// TIA Portal V17 export
// export: Created 2026-04-13T11:12:53.8543226Z, ExportSetting WithDefaults, DisplayName Totally Integrated Automation Portal, DisplayVersion V17 Update 4, DisplayName TIA Portal Openness, DisplayVersion V17 Update 4, DisplayName TIA Portal Version Control Interface, DisplayVersion V17, DisplayName SINAMICS Startdrive Advanced, DisplayVersion V17, DisplayName SINAMICS Startdrive G130, G150, S120, S150, SINAMICS MV, S210, DisplayVersion V17, DisplayName SINAMICS Startdrive G110M, G120, G120C, G120D, G120P, G115D, DisplayVersion V17, DisplayName STEP 7 Professional, DisplayVersion V17 Update 4, DisplayName STEP 7 Safety, DisplayVersion V17, DisplayName WinCC Professional, DisplayVersion V17 Update 4
TagTable "PW"
  PW_PH批号输入 : Int  (PLC tag PW.PH批号输入, HMI_连接_1, 1 s)
  PW_MS模式设定 : Real  (PLC tag PW.MS模式设定, HMI_连接_1, 1 s)
  PW_AQ安全停机 : Bool  (PLC tag PW.AQ安全停机, HMI_连接_1, 1 s)
  PW_自动运行报警 : Bool  (PLC tag PW.自动运行报警, HMI_连接_1, 1 s)
  PW_自动停止 : Bool  (PLC tag PW.自动停止, HMI_连接_1, 1 s)
  PW_MS模式状态 : Int  (PLC tag PW.MS模式状态, HMI_连接_1, 1 s)
  PW_ZT总通路 : Int  (PLC tag PW.ZT总通路, HMI_连接_1, 1 s)
